// Mitsubishi GX Works2 project: 04-06-2020 Timer   PLC: FX3U/FX3UC

PROGRAM MAIN
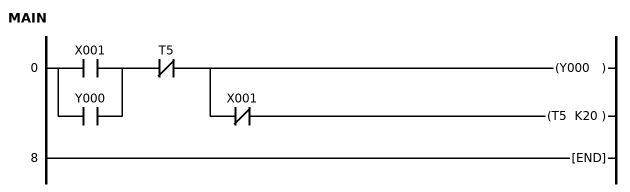
0     LD      X001
      OR      Y000
      ANI     T5
      OUT     Y000
      ANI     X001
      OUT     T5 K20
8     END
END_PROGRAM
